(* CoDeSys 2.3 export: BUTTONTRIGGEREDSCENE.EXP *)

(* POU Components/Scene/ButtonTriggeredScene, ST *)
FUNCTION_BLOCK ButtonTriggeredScene
VAR_INPUT
	input:BOOL;
END_VAR
VAR_OUTPUT
	a:BOOL;
	b:BOOL;
END_VAR
VAR
	Button:Button;
END_VAR
VAR_IN_OUT
	Scene:Scene;
END_VAR
button(input:=input);
scene(rotate:= button.longPressed, switch:= button.fallingEdge);
a:= scene.number = 1 OR scene.number = 2;
b:= scene.number = 1 OR scene.number = 3;
END_FUNCTION_BLOCK
